// TIA Portal V19 export
FUNCTION "FC_fPosfreePos" : Void   // FC128, STL
{ S7_Optimized_Access := 'FALSE' }
// stored: AutoNumber false
   VAR_INPUT
      WT_Nr : Int;
      WT_Typ : Byte;
      TypChk : Bool;
   END_VAR
   VAR_OUTPUT
      free : Bool;
      fPosfree : Bool;
      Zwangsziel : Int;
   END_VAR
   VAR_IN_OUT
      Ziel_1 : Int;
      leng_1 : Int;
      Ziel_2 : Int;
      leng_2 : Int;
      Reihe : Byte;
   END_VAR
   VAR_TEMP
      savAR1 : DWord;
      savAR2 : DWord;
      WT_DB : Word;
      ChkPos : Int;
      Adresse : DWord;
      BadTyp : Byte;
      PosTyp : Byte;
      TmpReihe : Byte;
      ZwZiel : Int;
      Leerzeit : Int;
      TmpZiel : Int;
      MemChk : Bool;
      Restzeit : DInt;
      nx_fposfree : Bool;
      temp_Free : Bool;
   END_VAR
BEGIN

NETWORK
TITLE = Register retten
// --------------------------------
// Register retten
// --------------------------------
      TAR1;
      T     #savAR1;
      TAR2;
      T     #savAR2;

NETWORK
TITLE = Initialisierung
      SET;
      S     #temp_Free;
      R     #fPosfree;
      R     #nx_fposfree;

      L     0;
      T     #Zwangsziel;
      T     #ZwZiel;
      T     #Leerzeit;
      T     #TmpZiel;

////// !!!!!!!!!!!!!!!!!!!!!!!!!!  !!!!!!!!!!!!
////// !!!!!!!!!!!!!!!!!!!!!!!!!!  !!!!!!!!!!!!
//Schleife evtl verbessern indem in Gruppen
//nach längster Leerzeit gesucht wird
////// !!!!!!!!!!!!!!!!!!!!!!!!!!  !!!!!!!!!!!!
////// !!!!!!!!!!!!!!!!!!!!!!!!!!  !!!!!!!!!!!!


NETWORK
TITLE = 
      L     #Ziel_1;
      L     "DB_POS".LENG;
      *I;
      L     "DB_POS".Offset;
      +I;
      SLD   3;
      LAR1;
      OPN   "DB_POS";
      L     DBB [AR1, P#0.0];  //"DB_POS".POS[0].Typ
      T     #BadTyp;
      L     5;  //Speichertest
      ==I;
      =     #MemChk;

retG: L     0;
      L     #leng_1;
      >=I;
      JC    nexG;
      +     -1;
      T     #leng_1;

      L     #Ziel_1;
      L     #leng_1;
      +I;
      T     #ChkPos;

      L     #ChkPos;
      L     "DB_POS".LENG;
      *D;
      L     "DB_POS".Offset;
      +D;
      SLD   3;
      LAR1;
      OPN   "DB_POS";
      L     DBB [AR1, P#0.0];  //"DB_POS".POS[0].Typ
      L     #BadTyp;  //nicht gleichen Typgruppe
      <>I;
      JC    retG;

      L     #WT_Nr;  //selbst gefunden
      L     DBB [AR1, P#36.0];  //next_WT
      ==I;
      O(;
      L     DBB [AR1, P#36.0];  //next_WT
      L     0;
      ==I;
      );
      AN    DBX [AR1, P#7.0];  //Sperre_in
      AN    DBX [AR1, P#9.1];  //notFGin
      A     DBX [AR1, P#9.3];  //FG_Posfree
      =     #nx_fposfree;

      L     0;  //Pos ist leer --> prüfen
      L     DBB [AR1, P#36.0];  //next_WT
      ==I;
      O     DBX [AR1, P#10.4];  //"DB_POS".POS[0].ignor_fPosFree
      AN    DBX [AR1, P#7.0];  //Sperre_in
      AN    DBX [AR1, P#9.1];  //notFGin
      JC    fnd;

      L     DBB [AR1, P#0.0];  //"DB_POS".POS[0].Typ
      L     0;
      ==I;
      A     DBX [AR1, P#9.1];  //notFGin
      O     DBX [AR1, P#7.0];  //Sperre_in
      JC    retG;

      L     #WT_Nr;  //selbst gefunden
      L     DBB [AR1, P#36.0];  //next_WT
      ==I;
      JC    fnd;
      JU    retG;

fnd:  OPN   "DB_POS";
      L     DBB [AR1, P#11.0];  //"DB_POS".POS[0].TrommelPos
      T     #PosTyp;

      L     #WT_Typ;  //Hi-Nibble prüfen vom WT
      AW    16#00F0;
      JZ    hiok;

      L     #PosTyp;
      AW    16#00F0;
      JZ    hiok;
      <>I;
      JC    retG;

hiok: AN    #TypChk;
      JC    WTYP;

      L     #WT_Typ;  //Lo-Nibble prüfen vom WT
      AW    16#000F;
      JZ    WTYP;

      L     #PosTyp;
      AW    16#000F;
      JZ    WTYP;
      <>I;
      JC    retG;

//-------------------------------------------
//Position reservieren
//-------------------------------------------
WTYP: A     #MemChk;
      JC    frst;
      AN    #temp_Free;
      S     #temp_Free;
      JC    frst;

      L     0;
      L     #Reihe;
      ==I;
      JC    LZC;

//------------------------------------------------
//neue Pos gleiche Reihe gemerkte Pos andere Reihe
// --> übernehmen neue Pos
//------------------------------------------------
      L     #Reihe;
      L     DBB [AR1, P#4.0];  //"DB_POS".POS[0].Reihe
      ==I;
      A(;
      L     #TmpReihe;
      L     #Reihe;
      <>I;
      );
      JC    frst;
//------------------------------------------------
//neue Pos andere Reihe gemerkte Pos gleiche Reihe
// --> übernehmen neue Pos
//------------------------------------------------
      L     #Reihe;
      L     DBB [AR1, P#4.0];  //"DB_POS".POS[0].Reihe
      <>I;
      A(;
      L     #TmpReihe;
      L     #Reihe;
      ==I;
      );
      JC    retG;
//------------------------------------------------
//bei gleichen Reihen Leerzeit berücksichtigen
//------------------------------------------------
LZC:  L     DBW [AR1, P#98.0];  //"DB_POS".POS[0].Leerzeit
      L     #Leerzeit;
      <=D;
      JC    retG;

frst: L     DBW [AR1, P#98.0];  //"DB_POS".POS[0].Leerzeit
      T     #Leerzeit;
      L     DBB [AR1, P#4.0];  //"DB_POS".POS[0].Reihe
      T     #TmpReihe;

      L     #ChkPos;
      T     #TmpZiel;
      SLD   3;
      T     #Adresse;
      OPN   "DB_Zwangsziel";
      L     0;
      L     DBB [#Adresse];
      ==I;
      T     #ZwZiel;

      A     #MemChk;
      JC    Take;

nexG: L     #Ziel_2;
      L     0;
      <>I;
      JC    wtr;
      A     #temp_Free;
      JC    Take;

      A     #nx_fposfree;
      =     #fPosfree;
      JU    raus;

wtr:  L     #Ziel_2;
      T     #Ziel_1;
      L     #leng_2;
      T     #leng_1;
      L     0;
      T     #Ziel_2;
      T     #leng_2;
      JU    retG;

Take: L     #ChkPos;
      L     "DB_POS".LENG;
      *D;
      L     "DB_POS".Offset;
      +D;
      SLD   3;
      LAR1;
      OPN   "DB_POS";
//Pos mit anderem WT belegt --> Abbruch
      L     DBB [AR1, P#36.0];
      L     #WT_Nr;
      <>I;
      A(;
      L     DBB [AR1, P#36.0];
      L     0;
      <>I;
      );
      R     #fPosfree;
      JC    raus;

//Pos gesperrt --> Abbruch
      L     DBB [AR1, P#0.0];  //PosTyp
      L     10;  //Typ QT
      <>I;
      A     DBX [AR1, P#9.1];  //notFG_in
      O     DBX [AR1, P#7.0];  //Sperre_in
      R     #fPosfree;
      JC    raus;

      L     0;
      L     DBB [AR1, P#36.0];
      <>I;
      JC    bel;
      L     #WT_Nr;
      T     DBB [AR1, P#36.0];

bel:  A     DBX [AR1, P#9.3];  //FG_Posfree
      AN    DBX [AR1, P#10.4];  //"DB_POS".POS[0].ignor_fPosFree
      AN    DBX [AR1, P#7.2];  //Sperre_out
      =     #fPosfree;

      L     #ZwZiel;
      T     #Zwangsziel;
      L     #TmpReihe;
      T     #Reihe;


NETWORK
TITLE = Adressregister wiederherstellen
//--------------------------------------
//Adressregister wiederherstellen
//--------------------------------------
raus: L     #savAR1;
      LAR1;
      L     #savAR2;
      LAR2;

NETWORK
TITLE = Ausgänge umkopieren
      A     #temp_Free;
      =     #free;

END_FUNCTION
